# EPICS autosave request: ipApp/Db/HP_Agilent_PS66xxA_settings.req
$(P)$(R)ReadAll.SCAN
$(P)$(R)SP_V_tweak
$(P)$(R)SP_C_tweak
